(* IEC 61131-3 sources: Faster/src/Ar/Faster, 3 files *)

(* ---- Types.typ ---- *)
(*
 * File: Types.typ
 * Copyright (c) 2023 Loupe
 * https://loupe.team
 *
 * This file is part of Faster, licensed under the MIT License.
 *)
TYPE

END_TYPE

(* ---- faster.fun ---- *)
(*
 * File: faster.fun
 * Copyright (c) 2023 Loupe
 * https://loupe.team
 *
 * This file is part of Faster, licensed under the MIT License.
 *)
{REDUND_ERROR} FUNCTION fasterInit : DINT (* *) (*$GROUP=User,$CAT=User,$GROUPICON=User.png,$CATICON=User.png*)
	VAR_INPUT
		pTimeStamps : UDINT;
		pTimeDeltas : UDINT;
		pSampleName : UDINT;
		maxSamples : DINT;
	END_VAR
END_FUNCTION

{REDUND_ERROR} FUNCTION fasterReset : DINT (* *) (*$GROUP=User,$CAT=User,$GROUPICON=User.png,$CATICON=User.png*)
END_FUNCTION

FUNCTION fasterStart : DINT
END_FUNCTION

{REDUND_ERROR} FUNCTION fasterTimeSinceLast : DINT (* *) (*$GROUP=User,$CAT=User,$GROUPICON=User.png,$CATICON=User.png*)
	VAR_INPUT
		label : STRING[FASTER_NAME_LENGTH];
	END_VAR
END_FUNCTION

{REDUND_ERROR} FUNCTION fasterTimeSinceLabel : DINT (* *) (*$GROUP=User,$CAT=User,$GROUPICON=User.png,$CATICON=User.png*)
	VAR_INPUT
		previous : STRING[FASTER_NAME_LENGTH];
		label : STRING[FASTER_NAME_LENGTH];
	END_VAR
END_FUNCTION

(* ---- Constants.var ---- *)
(*
 * File: Constants.var
 * Copyright (c) 2023 Loupe
 * https://loupe.team
 *
 * This file is part of Faster, licensed under the MIT License.
 *)
VAR CONSTANT
	FASTER_INTERNAL_SAMPLES : USINT := 100;
	FASTER_NAME_LENGTH : USINT := 80;
END_VAR
